Omron CX-Programmer project NewProject (CX-Programmer 9.73)

# PLC NewPLC1: CP1E N30

## Program NewProgram1 (cyclic task 0)

### Section Section1

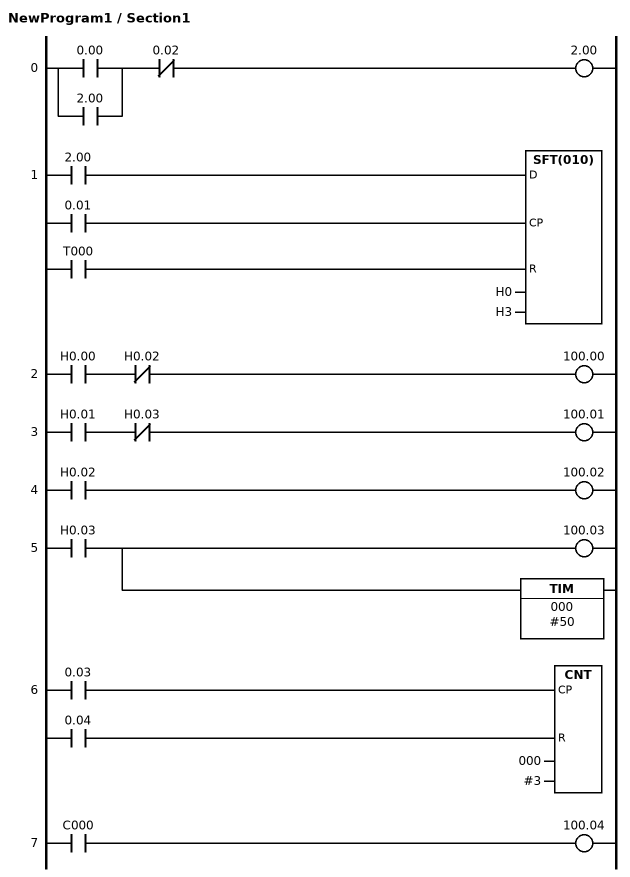
; rung 0
LD 0.00
OR 2.00
ANDNOT 0.02
OUT 2.00
; rung 1
LD 2.00
LD 0.01
LD T000
SFT(010) H0 H3
; rung 2
LD H0.00
ANDNOT H0.02
OUT 100.00
; rung 3
LD H0.01
ANDNOT H0.03
OUT 100.01
; rung 4
LD H0.02
OUT 100.02
; rung 5
LD H0.03
OUT 100.03
TIM 000 #50
; rung 6
LD 0.03
LD 0.04
CNT 000 #3
; rung 7
LD C000
OUT 100.04

### Section END
; rung 0
END(001)